// Common contract every FB_Alarm* exposes. Lets HMI gateways and aggregators
// acknowledge a heterogeneous collection of alarms uniformly.
INTERFACE I_Alarm

METHOD Ack : E_RpcMethodResponse
VAR_INPUT
    eRequester : E_Requester := E_Requester.PROG;
END_VAR
END_METHOD

METHOD LockSource : E_RpcMethodResponse
VAR_INPUT
    bLock : BOOL;
END_VAR
END_METHOD

END_INTERFACE

(* stored: Version 1.1.0.1, ProductVersion 3.1.4026.12
   Itf I_Alarm: Id {c0000006-0000-0000-0000-000000000001}
   Method Ack: Id {c0000006-0000-0000-1000-000000000001}
   Method LockSource: Id {c0000006-0000-0000-1000-000000000002} *)
